FUNCTION ARR08X_TO_BOOLS (* this Function extracts the 8 BOOLS from a 8-BOOL Array *)
  (* Standard: 61499-1; Description: Copyright (c) 2024 HR Agrartechnik GmbH This program and the accompanying materials are made available under the terms of the Eclipse Public License 2.0 which is available at https://www.eclipse.org/legal/epl-2.0/ SPDX-License-Identifier: EPL-2.0 *)
  (* Version 1.0, 2024-02-22, Franz Höpfinger, HR Agrartechnik GmbH *)
  PACKAGE logiBUS::utils::conversion::arr::forwarding;
  IMPORT eclipse4diac::core::TypeHash;
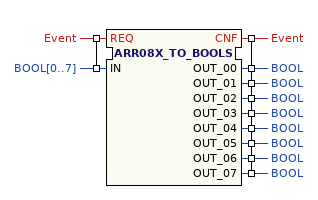
  EVENT_INPUT
    REQ WITH IN;
  END_EVENT
  EVENT_OUTPUT
    CNF WITH OUT_00, OUT_01, OUT_02, OUT_03, OUT_04, OUT_05, OUT_06, OUT_07;
  END_EVENT
  VAR_INPUT
    IN : ARRAY [0..7] OF BOOL; (* ARR08X Input *)
  END_VAR
  VAR_OUTPUT
    OUT_00 : BOOL; (* BIT 00 *)
    OUT_01 : BOOL; (* BIT 01 *)
    OUT_02 : BOOL; (* BIT 02 *)
    OUT_03 : BOOL; (* BIT 03 *)
    OUT_04 : BOOL; (* BIT 04 *)
    OUT_05 : BOOL; (* BIT 05 *)
    OUT_06 : BOOL; (* BIT 06 *)
    OUT_07 : BOOL; (* BIT 07 *)
  END_VAR
  BODY IN ST:
PACKAGE logiBUS::utils::conversion::arr::forwarding;

(* this Function extracts the 8 BOOLS from a 8-BOOL Array *)
FUNCTION ARR08X_TO_BOOLS

VAR_INPUT
	IN : ARRAY[0..7] OF BOOL; // ARR08X Input
END_VAR

VAR_OUTPUT
	OUT_00 : BOOL; // BIT 00
	OUT_01 : BOOL; // BIT 01
	OUT_02 : BOOL; // BIT 02
	OUT_03 : BOOL; // BIT 03
	OUT_04 : BOOL; // BIT 04
	OUT_05 : BOOL; // BIT 05
	OUT_06 : BOOL; // BIT 06
	OUT_07 : BOOL; // BIT 07
END_VAR

OUT_00 := IN[0];
OUT_01 := IN[1];
OUT_02 := IN[2];
OUT_03 := IN[3];
OUT_04 := IN[4];
OUT_05 := IN[5];
OUT_06 := IN[6];
OUT_07 := IN[7];

END_FUNCTION
  END_BODY
END_FUNCTION
